// TIA Portal V15 export
// export: Created 2018-05-29T12:25:38.1552518Z, ExportSetting WithDefaults, DisplayName Totally Integrated Automation Portal, DisplayVersion V15, DisplayName TIA Portal Openness, DisplayVersion V15, DisplayName STEP 7 Professional, DisplayVersion V15, DisplayName WinCC Professional, DisplayVersion V15
FUNCTION "EM_Instance_5_fc" : Void   // FC1, STL
TITLE = _fc
{ S7_Optimized_Access := 'TRUE' }
VERSION : 0.1
// test
// stored: AutoNumber true, UDAEnableTagReadback false
BEGIN

NETWORK
TITLE = Main
// comment:
// Call the EM FB with the corresponding DB instance
CALL EM_I_OUT, EM_Instance_5
	em_id := 30
	Pump_RUN := M104.QNOFF2
	Pump_QERR := M104.QERR
	Pump_EERR := M104.QERR_EXT
	FS01_PV := LS002.QON
	PIC01_PV := LIC005.PV
	PIC01_ERR := LIC005.QERR
	LT01_PV := LT005.QfVal
	LT01_AHH := LT005.LIM_Qb01
	LT01_AH := LT005.LIM_Qb02
	LT01_AL := LT005.LIM_Qb03
	LT01_ALL := LT005.LIM_Qb04
	LT01_ERR := LT005.QERR
	BV_Bottom_OPN := MV005.QOPEN
	BV_Bottom_CLS := MV005.QCLOSE
	BV_Bottom_MERR := MV005.QMON_ERR
	BV_Tran_M04_OPN := MV003.QOPEN
	BV_Tran_M04_CLS := MV003.QCLOSE
	BV_Tran_M04_MERR := MV003.QMON_ERR
	Pump_ON := M104.L_ON
	Pump_AUT := M104.L_AUT
	PIC01_EXT := LIC005.L_REMOTE
	PIC01_SP := LIC005.HMI_SP_INT
	PIC01_AUT := LIC005.L_AUT
	PIC01_VAL_OUT := LIC005.HMI_MAN
	PIC01_SET_SP := LIC005.Set_SP
	PIC01_SET_OUT := LIC005.Set_Output
	BV_Bottom_CMD := MV005.AUT_OP
	BV_Tran_M04_CMD := MV003.AUT_OP
END_FUNCTION
